(* IEC 61131-3 sources: CS_4_Aufzugsteuerung/src/Stations/CP112/Steuerung/Class/clsEmgStop_1, 1 file *)

(* ---- clsEmgStop_1.st ---- *)
(*!
<Class
	Name               = "clsEmgStop_1"
	Revision           = "0.0"
	RealtimeTask       = "true"
	CyclicTask         = "false"
	BackgroundTask     = "false"
	Sigmatek           = "false"
	OSInterface        = "false"
	HighPriority       = "false"
	Automatic          = "false"
	UpdateMode         = "Prescan"
	SharedCommandTable = "true"
	Objectsize         = "(284,120)">
	<Channels>
		<Server Name="ClassSvr" Visualized="false" Initialize="false" WriteProtected="true" Retentive="false"/>
		<Server Name="sVisuNotStop" Visualized="true" Remotely="true" Initialize="false" WriteProtected="true" Retentive="false"/>
		<Client Name="c1" Required="true" Internal="false"/>
		<Client Name="c2" Required="true" Internal="false"/>
	</Channels>
</Class>
*)
clsEmgStop_1 : CLASS
  //Servers:
	ClassSvr 	: SvrChCmd_DINT;
	sVisuNotStop 	: SvrCh_DINT;
  //Clients:
	c1 	: CltCh_DINT;
	c2 	: CltCh_DINT;
  //Variables:
		xEmgStop 	: BOOL;
  //Functions:

	FUNCTION VIRTUAL GLOBAL RtWork
		VAR_INPUT
			EAX 	: UDINT;
		END_VAR
		VAR_OUTPUT
			state (EAX) 	: UDINT;
		END_VAR;

	FUNCTION GLOBAL EmgStop
		VAR_OUTPUT
			xOut 	: BOOL;
		END_VAR;
  //Tables:
	FUNCTION @STD
		VAR_OUTPUT
			ret_code	: CONFSTATES;
		END_VAR;
	FUNCTION GLOBAL TAB @CT_;
END_CLASS;

FUNCTION VIRTUAL GLOBAL clsEmgStop_1::RtWork
	VAR_INPUT
		EAX 	: UDINT;
	END_VAR
	VAR_OUTPUT
		state (EAX) 	: UDINT;
	END_VAR

  //IO uebergeben
  c1 := c1.Read();
  c2 := c2.Read();

  //HMI uebergeben
  sVisuNotStop := xEmgStop;

  // monitoring
  IF (c1 = 1) AND (c2 = 1) THEN
    xEmgStop := FALSE;
  ELSE
    xEmgStop := TRUE;
  END_IF;

	state := READY;

END_FUNCTION

FUNCTION GLOBAL clsEmgStop_1::EmgStop
	VAR_OUTPUT
		xOut 	: BOOL;
	END_VAR

  //uebergabe an Methodenaufrud

 xOut := xEmgStop;

END_FUNCTION
